FUNCTION F_STRINGSPLIT : ARRAY[0..Parameters.iSplitArraySize] OF STRING(255)
VAR_INPUT
	sInput			: STRING(255);
	sSplitChar		: STRING(1);
END_VAR
VAR
	sCopy			: STRING(255);
	sSplit			: STRING(255);
	iDeleteLen		: INT;
	i				: INT;
END_VAR

sCopy := sInput;

FOR i := 0 TO Parameters.iSplitArraySize DO
	IF FIND(sCopy, sSplitChar) > 0 THEN
		sSplit := LEFT(sCopy, FIND(sCopy, sSplitChar) - 1);
		iDeleteLen := LEN(sSplit) + LEN(sSplitChar);
	ELSE
		sSplit := sCopy;
		iDeleteLen := LEN(sSplit);
	END_IF
	
	// Take the string value
	F_STRINGSPLIT[i] := sSplit;
	
	// Delete 
	sCopy := DELETE(sCopy, iDeleteLen, 1);
	
	// End of split
	IF sCopy = '' THEN
		EXIT;
	END_IF
END_FOR

END_FUNCTION

(* stored: Version 1.1.0.1, ProductVersion 3.1.4024.9
   POU F_STRINGSPLIT: Id {bf09d747-8a2c-4de8-9a8b-909da6c686c1}, SpecialFunc None *)
